TYPE "Prod_Halted_Str"
VERSION : 0.1
// Block: Prod_Halted_Str
   STRUCT
      Code : Int;
      Detail : String;
   END_STRUCT;

END_TYPE
